(* CoDeSys 2.3.9.48 project: 20170405_WUR.pro *)
(* Version: 0.9 *)
(* Description: Project Distributie Automatisering *)
(* Libraries: Serial_Interface_01.lib 22.4.13 12:50:14, Util.lib 30.1.13 13:05:12, WagoLib787_01.lib 10.11.14 13:02:32, mod_com.lib 30.1.13 13:05:12, WagoConfigToolLIB.lib 30.1.13 13:05:12, C:\Program Files\WAGO Software\CODESYS V2.3\Targets\WAGO\Libraries\32_Bit\PowerMeasurement_495_02.lib*5.4.17 15:41:49, SysLibTime.lib 30.1.13 13:05:12, SerComm.lib 30.1.13 13:05:12, SysLibSockets.lib 22.5.14 16:16:32, SysLibFile.lib 30.1.13 13:05:12, C:\Program Files\WAGO Software\CODESYS V2.3\Targets\WAGO\Libraries\32_Bit\Ethernet.lib*5.4.17 15:41:49, SysLibMem.lib 30.1.13 13:05:12, SysLibSem.lib 30.1.13 13:05:12, SysLibRtc.lib 30.1.13 13:05:12, WagoLibEthernet_01.lib 1.4.15 14:24:28, WAGOLIBNTP.lib*19.8.11 14:53:14, Modb_l05.lib 13.5.15 10:30:08, SysLibDir.lib 30.1.13 13:05:12, C:\Program Files\WAGO Software\CODESYS V2.3\Targets\WAGO\Libraries\32_Bit\WAGO_Datalogger_02.lib*5.4.17 15:41:49, Wago_MBCFG_SERIAL_01.lib*1.4.15 14:24:28, Wago_MBCFG_COMMON_01.lib 1.4.15 14:24:28, Standard.lib 20.5.14 08:13:26, Iecsfc.lib 30.1.13 13:05:12, SYSLIBCALLBACK.LIB 30.1.13 13:05:12 *)

(* Task configuration *)
TASK WriteData (PRIORITY := 31); (* freewheeling *)
	WRITE_DATA();
END_TASK
TASK Measurements (PRIORITY := 1, INTERVAL := T#100ms);
	PQ_1();
END_TASK

(* Global variable list: Global_Variables *)
VAR_GLOBAL

	arMeasurementsGroup1					:	ARRAY[1.. iNumberMeasurementVar] OF REAL;
	arSystemState		AT %MW0			:	ARRAY[1.. iNumberSystemVar] OF REAL; 			(* Array containing all the system parameters. Values are accessable through modbus tcp starting from register 12288. REAL uses two registers per variable *)

END_VAR

VAR_GLOBAL CONSTANT

(* Read / write CSV-files *)
	iMaxParams			:	INT:=8;(* Number of Parameters per File *)
	gc_ParameterCount	:	INT:=1;(* Number of Values per Parameter *)
	gc_RawDataSize		:	UINT:=500; (* Raw data size for reading in file ASCII *)
	gcRowExcel			:	INT:=1;

	iNumberMeasurementVar	:	INT := 20;
	iNumberSystemVar			:	INT := 200;


END_VAR

VAR_GLOBAL PERSISTENT RETAIN

	CurrentRatioPQ1						:	WORD := 400;			(* Current transformer ratio, eg 5 A / 400 A *)
	CurrentRatioPQ2						:	WORD := 400;

END_VAR

(* Data type *)
TYPE typCSV :
STRUCT
	sDescription	:STRING;
	Parameter		:ARRAY[1..gc_ParameterCount] OF STRING;
END_STRUCT
END_TYPE

(* POU WRITE_CSV/WRITE_DATA, FBD *)
PROGRAM WRITE_DATA
VAR
	FB1				: FbDatalogger;
	xGo				: BOOL		:= TRUE;
	xTrigger			: BOOL;
	Channels			: ARRAY [1.. 80] OF typUserInput;
	Settings			: typConfigDatalogger;
	bDType			: BYTE := 1;
	xFirstCycle			: BOOL := TRUE;
	i: INT;

END_VAR
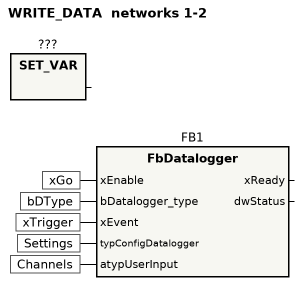
_FBD_ (* Function Block Diagram *)
NETWORK 1
	???:SET_VAR()
NETWORK 2
	FB1:FbDatalogger(xEnable: xGo, bDatalogger_type: bDType, xEvent: xTrigger, typConfigDatalogger: Settings, atypUserInput: Channels)
_END_FBD_
(* the same logic as Structured Text *)
(* Network 1: see the listing above *)
(* Network 2 *)
FB1(xEnable := xGo, bDatalogger_type := bDType, xEvent := xTrigger, typConfigDatalogger := Settings, atypUserInput := Channels);
END_PROGRAM
ACTION SET_VAR:
IF xFirstCycle THEN

	settings.bInterval					:= 3; 						(* 1 = hour, 2= minutes, 3 = seconds *)
	settings.iIntervalFactor			:= 5;						(* number of hours/minutes/seconds, depending on choice b.Interval *)
	settings.sFilename				:= 'Meetdata.csv';				(* Filename csv-file *)
	settings.sPath						:= '/media/sd/';				(* Path where the csv-file is stored *)
	settings.xAppendDate			:= TRUE;					(* When true, the date on the controller is added to the filename*)
	settings.xCyclicLogging			:= TRUE;					(* When true, information is stored cyclic on the controller/SD card *)

	Channels[1].xChannelExists		:= TRUE;
	Channels[1].sChannelName		:= 'PhaseCurrentl2';
	Channels[1].sUnit					:= 'A';
	Channels[1].rAlarmLowerLimit	:= -10000000;
	Channels[1].rAlarmUpperLimit	:= 10000000;

	Channels[2].xChannelExists		:= TRUE;
	Channels[2].sChannelName		:= 'VoltageV31';
	Channels[2].sUnit					:= 'V';
	Channels[2].rAlarmLowerLimit	:= -10000000;
	Channels[2].rAlarmUpperLimit	:= 10000000;

	Channels[3].xChannelExists		:= TRUE;
	Channels[3].sChannelName		:= 'Pactive';
	Channels[3].sUnit					:= 'W';
	Channels[3].rAlarmLowerLimit	:= -10000000;
	Channels[3].rAlarmUpperLimit	:= 10000000;

	Channels[4].xChannelExists		:= TRUE;
	Channels[4].sChannelName		:= 'Preactive';
	Channels[4].sUnit					:= 'VAr';;
	Channels[4].rAlarmLowerLimit	:= -10000000;
	Channels[4].rAlarmUpperLimit	:= 10000000;

	Channels[5].xChannelExists		:= TRUE;
	Channels[5].sChannelName		:= 'ShortCircuitDirectionA';
	Channels[5].sUnit					:= ' ';
	Channels[5].rAlarmLowerLimit	:= -10000000;
	Channels[5].rAlarmUpperLimit	:= 10000000;

	Channels[6].xChannelExists		:= TRUE;
	Channels[6].sChannelName		:= 'ShortCircuitDirectionB';
	Channels[6].sUnit					:= ' ';
	Channels[6].rAlarmLowerLimit	:= -10000000;
	Channels[6].rAlarmUpperLimit	:= 10000000;

	Channels[7].xChannelExists		:= TRUE;
	Channels[7].sChannelName		:= 'Phase1';
	Channels[7].sUnit					:= ' ';
	Channels[7].rAlarmLowerLimit	:= -10000000;
	Channels[7].rAlarmUpperLimit	:= 10000000;

	Channels[8].xChannelExists		:= TRUE;
	Channels[8].sChannelName		:= 'Phase2';
	Channels[8].sUnit					:=  ' ';
	Channels[8].rAlarmLowerLimit	:= -10000000;
	Channels[8].rAlarmUpperLimit	:= 10000000;

	Channels[9].xChannelExists		:= TRUE;
	Channels[9].sChannelName		:= 'Phase3';
	Channels[9].sUnit					:=  ' ';
	Channels[9].rAlarmLowerLimit	:= -10000000;
	Channels[9].rAlarmUpperLimit	:= 10000000;

	Channels[10].xChannelExists		:= TRUE;
	Channels[10].sChannelName		:= 'StatusRemoteSwitching';
	Channels[10].sUnit					:=  ' ';
	Channels[10].rAlarmLowerLimit	:= -10000000;
	Channels[10].rAlarmUpperLimit	:= 10000000;


	Channels[11].xChannelExists		:= TRUE;
	Channels[11].sChannelName		:= 'SwitchLoadBreaker';
	Channels[11].sUnit					:=  ' ';
	Channels[11].rAlarmLowerLimit	:= -10000000;
	Channels[11].rAlarmUpperLimit	:= 10000000;

	Channels[12].xChannelExists		:= TRUE;
	Channels[12].sChannelName		:= 'Bay3CurrentL1';
	Channels[12].sUnit					:=  'A ';
	Channels[12].rAlarmLowerLimit	:= -10000000;
	Channels[12].rAlarmUpperLimit	:= 10000000;

	Channels[13].xChannelExists		:= TRUE;
	Channels[13].sChannelName		:= 'Bay3CurrentL2';
	Channels[13].sUnit					:=  'A ';
	Channels[13].rAlarmLowerLimit	:= -10000000;
	Channels[13].rAlarmUpperLimit	:= 10000000;

	Channels[14].xChannelExists		:= TRUE;
	Channels[14].sChannelName		:= 'Bay3CurrentL3';
	Channels[14].sUnit					:=  'A ';
	Channels[14].rAlarmLowerLimit	:= -10000000;
	Channels[14].rAlarmUpperLimit	:= 10000000;

	Channels[15].xChannelExists		:= TRUE;
	Channels[15].sChannelName		:= 'Bay4CurrentL1';
	Channels[15].sUnit					:=  'A ';
	Channels[15].rAlarmLowerLimit	:= -10000000;
	Channels[15].rAlarmUpperLimit	:= 10000000;

	Channels[16].xChannelExists		:= TRUE;
	Channels[16].sChannelName		:= 'Bay4CurrentL2';
	Channels[16].sUnit					:=  'A ';
	Channels[16].rAlarmLowerLimit	:= -10000000;
	Channels[16].rAlarmUpperLimit	:= 10000000;

	Channels[17].xChannelExists		:= TRUE;
	Channels[17].sChannelName		:= 'Bay4CurrentL3';
	Channels[17].sUnit					:=  'A ';
	Channels[17].rAlarmLowerLimit	:= -10000000;
	Channels[17].rAlarmUpperLimit	:= 10000000;

	xFirstCycle := FALSE;

END_IF

	Channels[1].rValue			:= MBCFG_ModbusSlave.PhaseCurrenL2;
	Channels[2].rValue			:= MBCFG_ModbusSlave.VoltageV31;
	Channels[3].rValue			:= MBCFG_ModbusSlave.Pactive;
	Channels[4].rValue			:= MBCFG_ModbusSlave.Preactive;
	Channels[5].rValue			:= MBCFG_ModbusSlave.ShortCircuitA;
	Channels[6].rValue			:= MBCFG_ModbusSlave.ShortCircuitB;
	Channels[7].rValue			:= MBCFG_ModbusSlave.Phase1;
	Channels[8].rValue			:= MBCFG_ModbusSlave.Phase2;
	Channels[9].rValue			:= MBCFG_ModbusSlave.Phase3;
	Channels[10].rValue			:= MBCFG_ModbusSlave.StatusRemoteSwitching;
	Channels[11].rValue			:= MBCFG_ModbusSlave.SwitchLoadBreaker;
	Channels[12].rValue			:= PQ_1.arCurrent[1];
	Channels[13].rValue			:= PQ_1.arCurrent[2];
	Channels[14].rValue			:= PQ_1.arCurrent[3];
	Channels[15].rValue			:= PQ_2.arCurrent[1];
	Channels[16].rValue			:= PQ_2.arCurrent[2];
	Channels[17].rValue			:= PQ_2.arCurrent[3];





(* For-loop to set the channels to be written on the SD-card *)
END_ACTION

(* POU PQ/PQ_1, FBD *)
PROGRAM PQ_1
VAR
	abProcessImageInput	AT %IW48				: ARRAY[0..23] OF BYTE;
	abProcessImageOutput 	AT %QW48 			: ARRAY[0..23] OF BYTE;

	bToken										: BYTE;

	State_750_495 							: Fb_750_495_State;
		typ_750_495_State 						: typ_750_495_State;

	Configuration_750_495					: Fb_750_495_Configuration;
		typConfig_750_495						: typConfig_750_495;
		xReadyConfig								: BOOL;
		bFeedbackConfig							: BYTE;

	AC_Compact_01_750_495				: Fb_750_495_AC_Compact_01;
		rTotalActivePower							: REAL;
		rTotalReactivePower						: REAL;
		rTotalApparentPower						: REAL;
		rTotalPowerFactorPF						: REAL;
		rTotalActiveEnergy							: REAL;
		rTotalReactiveEnergy						: REAL;
		rTotalApparentEnergy						: REAL;
		rCurrentN									: REAL;
		xRotatingField								: BOOL;
		arCurrent									: ARRAY[1..3] OF REAL;
		axOvercurrent								: ARRAY[1..3] OF BOOL;
		arVoltage_L_N							: ARRAY[1..3] OF REAL;
		axUndervoltage							: ARRAY[1..3] OF BOOL;
		axOvervoltage								: ARRAY[1..3] OF BOOL;
		arActivePower								: ARRAY[1..3] OF REAL;
		arReactivePower							: ARRAY[1..3] OF REAL;
		arApparentPower							: ARRAY[1..3] OF REAL;
		arCosPhi									: ARRAY[1..3] OF REAL;
		arPowerFactorPF							: ARRAY[1..3] OF REAL;
		arFrequency								: ARRAY[1..3] OF REAL;
		axNoZero									: ARRAY[1..3] OF BOOL;
		axVoltSag									: ARRAY[1..3] OF BOOL;
		ai4Quadrant								: ARRAY[1..3] OF INT;

		xReadyCompact_01						: BOOL;
		abFeedbackCompact_01					: ARRAY[1..8] OF BYTE;


END_VAR
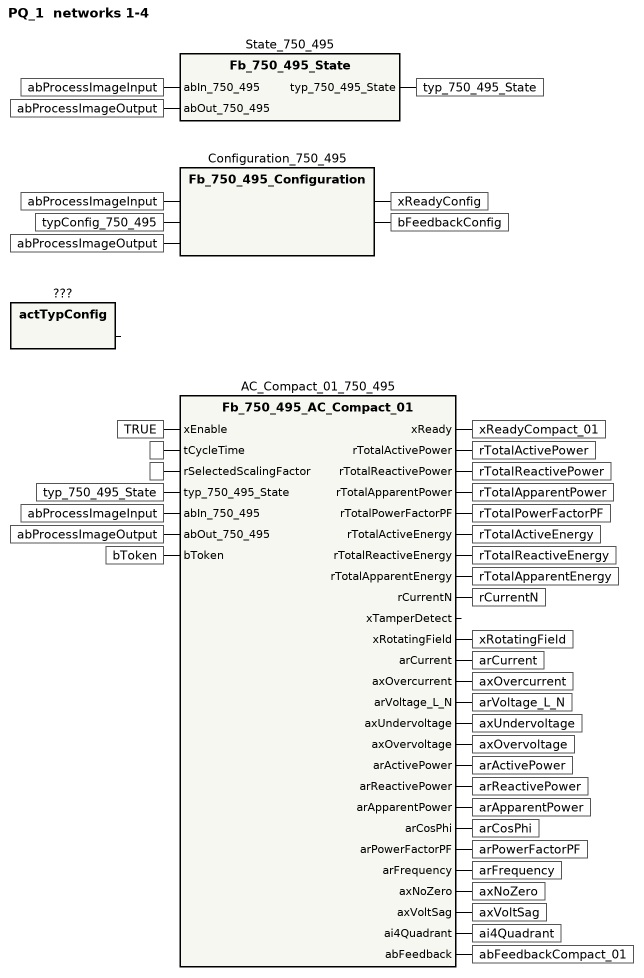
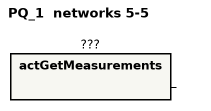
_FBD_ (* Function Block Diagram *)
NETWORK 1
	State_750_495:Fb_750_495_State(abIn_750_495: abProcessImageInput, abOut_750_495: abProcessImageOutput) => typ_750_495_State
NETWORK 2
	Configuration_750_495:Fb_750_495_Configuration(abProcessImageInput, typConfig_750_495, abProcessImageOutput, out 2 => bFeedbackConfig) => xReadyConfig
NETWORK 3
	???:actTypConfig()
NETWORK 4
	AC_Compact_01_750_495:Fb_750_495_AC_Compact_01(xEnable: TRUE, tCycleTime: , rSelectedScalingFactor: , typ_750_495_State: typ_750_495_State, abIn_750_495: abProcessImageInput, abOut_750_495: abProcessImageOutput, bToken: bToken, rTotalActivePower => rTotalActivePower, rTotalReactivePower => rTotalReactivePower, rTotalApparentPower => rTotalApparentPower, rTotalPowerFactorPF => rTotalPowerFactorPF, rTotalActiveEnergy => rTotalActiveEnergy, rTotalReactiveEnergy => rTotalReactiveEnergy, rTotalApparentEnergy => rTotalApparentEnergy, rCurrentN => rCurrentN, xRotatingField => xRotatingField, arCurrent => arCurrent, axOvercurrent => axOvercurrent, arVoltage_L_N => arVoltage_L_N, axUndervoltage => axUndervoltage, axOvervoltage => axOvervoltage, arActivePower => arActivePower, arReactivePower => arReactivePower, arApparentPower => arApparentPower, arCosPhi => arCosPhi, arPowerFactorPF => arPowerFactorPF, arFrequency => arFrequency, axNoZero => axNoZero, axVoltSag => axVoltSag, ai4Quadrant => ai4Quadrant, abFeedback => abFeedbackCompact_01) => xReadyCompact_01
NETWORK 5
	???:actGetMeasurements()
_END_FBD_
(* the same logic as Structured Text *)
(* Network 1 *)
State_750_495(abIn_750_495 := abProcessImageInput, abOut_750_495 := abProcessImageOutput);
typ_750_495_State := State_750_495.typ_750_495_State;
(* Network 2: see the listing above *)
(* Network 3: see the listing above *)
(* Network 4: see the listing above *)
(* Network 5: see the listing above *)
END_PROGRAM
ACTION actGetMeasurements:
arMeasurementsGroup1[1] := arVoltage_L_N[1];
arMeasurementsGroup1[2] := arVoltage_L_N[2];
arMeasurementsGroup1[3] := arVoltage_L_N[3];
arMeasurementsGroup1[4] := arCurrent[1];
arMeasurementsGroup1[5] := arCurrent[2];
arMeasurementsGroup1[6] := arCurrent[3];
END_ACTION
ACTION actTypConfig:
typConfig_750_495.typChannelConfig[1].xEnableUserScaling:= TRUE;
typConfig_750_495.typChannelConfig[1].wCurrentTransformerRatio :=CurrentRatioPQ1;

typConfig_750_495.typChannelConfig[2].xEnableUserScaling:= TRUE;
typConfig_750_495.typChannelConfig[2].wCurrentTransformerRatio :=CurrentRatioPQ1;

typConfig_750_495.typChannelConfig[3].xEnableUserScaling:= TRUE;
typConfig_750_495.typChannelConfig[3].wCurrentTransformerRatio :=CurrentRatioPQ1;

typConfig_750_495.xWriteConfig := TRUE;
END_ACTION

(* POU PLC_PRG, FBD *)
PROGRAM PLC_PRG
(*
  Function: 	Reading a CSV file
  Description: 	This project shows a functionblock which reads data from a CSV file into an array.
				Each line in the CSV contains a description and a real value.
				Each parameter  is terminated by CR LF.

---- Example CSV File -----

A_Value;245345
B_Value;0							
C_Value;8.3							
D_Value;-123439.3 						
E_Value;1						*)

VAR
	xLoad					: 	BOOL; (* Initiate load operation *)
	xSave					: 	BOOL; (* Initiate save operation *)
	sLoadStatus			: 	STRING; (* Feedback on load *)
	sSaveStatus			: 	STRING; (* Feedback on save *)
	ConfigData			: 	ARRAY [1..iMaxParams] OF  typCSV; (* Structure with the config data being loaded or saved *)
	sFileName			: 	STRING := 'config.csv'; (* Working Filename *)
	bSeperator 			: 	BYTE := 59; (* Semicolon (;) is the seperator between parameter and value. *)
	iError					: 	INT; (* Error Code for Save *)
	xWriteToSD			: 	BOOL := TRUE; (* User selectable location for file operation, on = 750-880 SD, off = internal flash *)
	sFilePath				: 	STRING; (* SD card is S:\, Internal Path is blank, but this points to the PLC folder *)
	sFilePath_Name		: 	STRING; (* Complete path + filename *)

	xReadFirstCycle		:	BOOL := TRUE;

	SetIPConfig				:	configToolFB;
	SetIP						:	configToolFB;
	SetSubnet					:	configToolFB;
	SetGateway				:	configToolFB;
	SetNTP					:	configToolFB;
	SetNTPEnable			:	configToolFB;
	SetSNMPName			:	configToolFB;
	SetSNMPDescription		:	configToolFB;
	SetSNMPLocation			:	configToolFB;
	SetSNMPContact			:	configToolFB;

	GetIPConfig				:	configToolFB;
	GetIP						:	configToolFB;
	GetSubnet					:	configToolFB;
	GetGateway				:	configToolFB;
	GetNTP					:	configToolFB;
	GetSNMPName			:	configToolFB;
	GetSNMPDescription		:	configToolFB;
	GetSNMPLocation		:	configToolFB;
	GetSNMPContact			:	configToolFB;
	GetFirmware				:	configToolFB;
	GetMACAddress			:	configToolFB;
	GetProjectDate			:	configToolFB;
	GetProjectDescription	:	configToolFB;
	GetProjectVersion			:	configToolFB;

	stSetIPConfigCallstring				:	STRING(80);
	stSetIPCallstring						:	STRING(80);
	stSetSubnetCallstring				:	STRING(80);
	stSetGatewayCallstring				:	STRING(80);
	stSetNTPCallstring					:	STRING(80);

	iSetIPConfigCallstringResult			:	INT;
	iSetIPCallstringResult				:	INT;
	iSetSubnetCallstringResult			:	INT;
	iSetGatewayCallstringResult			:	INT;
	iSetNTPCallstringResult				: 	INT;
	iSetNTPEnabledCallstringResult	:	INT;

	iGetIPConfigCallstringResult			:	INT;
	iGetIPCallstringResult				:	INT;
	iGetSubnetCallstringResult			:	INT;
	iGetGatewayCallstringResult			:	INT;
	iGetNTPCallstringResult				: 	INT;
	iGetNTPEnabledCallstringResult	:	INT;

	iGetFirmwareCallstringResult				:	INT;
	iGetMACAddressCallstringResult			:	INT;
	iGetProjectDateCallstringResult				:	INT;
	iGetProjectDescriptionCallstringResult		:	INT;
	iGetProjectVersionCallstringResult			:	INT;

	stGetIPConfigCallstring				:	STRING(80);
	stGetIPCallstring						:	STRING(80);
	stGetSubnetCallstring				:	STRING(80);
	stGetGatewayCallstring				:	STRING(80);
	stGetNTPCallstring					:	STRING(80);

	stSetIPConfigResult					:	STRING(80);
	stSetIPResult							:	STRING(80);
	stSetSubnetResult					:	STRING(80);
	stSetGatewayResult					:	STRING(80);
	stSetNTPResult						:	STRING(80);

	stGetIPConfigResult					:	STRING(80);
	stGetIPResult							:	STRING(80);
	stGetSubnetResult					:	STRING(80);
	stGetGatewayResult					:	STRING(80);
	stGetNTPResult						:	STRING(80);

	stSetSNMPNameDeviceCallstring					:	STRING(80);
	stSetSNMPDescriptionCallstring						:	STRING(80);
	stSetSNMPPhysicalLocationCallstring				:	STRING(80);
	stSetSNMPContactCallstring							:	STRING(80);

	stGetSNMPNameDeviceResult						:	STRING(80);
	stGetSNMPDescriptionResult						:	STRING(80);
	stGetSNMPPhysicalLocationResult					:	STRING(80);
	stGetSNMPContactResult							:	STRING(80);

	stGetFirmwareResult									:	STRING(80);
	stGetMACAddressResult								:	STRING(80);
	stGetProjectDateResult								:	STRING(80);
	stGetProjectDescriptionResult						:	STRING(80);
	stGetProjectVersionResult							:	STRING(80);

	iSetSNMPNameDeviceCallstringResult				:	INT;
	iSetSNMPDescriptionCallstringResult				:	INT;
	iSetSNMPPhysicalLocationCallstringResult			:	INT;
	iSetSNMPContactCallstringResult					:	INT;

	iGetSNMPNameDeviceCallstringResult				:	INT;
	iGetSNMPDescriptionCallstringResult				:	INT;
	iGetSNMPPhysicalLocationCallstringResult			:	INT;
	iGetSNMPContactCallstringResult					:	INT;

	CurrentTimeDate										:	STRING;

END_VAR
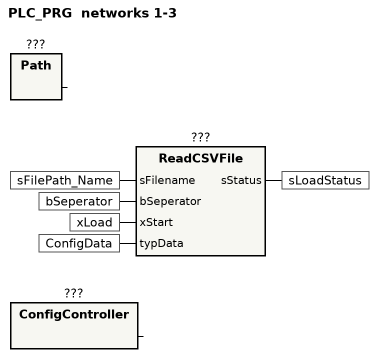
_FBD_ (* Function Block Diagram *)
NETWORK 1
	???:Path()
NETWORK 2
	???:ReadCSVFile(sFilename: sFilePath_Name, bSeperator: bSeperator, xStart: xLoad, typData: ConfigData) => sLoadStatus
NETWORK 3
	???:ConfigController()
_END_FBD_
END_PROGRAM
ACTION ConfigController:
IF xReadFirstCycle = TRUE THEN

	(*xLoad := TRUE;*)

	IF sLoadStatus = 'Data read OK' THEN
	
		(* Set Ethernet settings of controller *)
		
		(* Set static IP-Address*)
		
		
			SetIPConfig(
			bEnable:= TRUE,
			stCallString:= 'config_interfaces interface=X1 config-type=static state=enabled',
			stResultString=> stSetIPConfigResult,
			iFbResult=> iSetIPCallstringResult );
		
		(* Set IP-Address of controller *)
		
			stSetIPCallstring := CONCAT('config_interfaces interface X1 ip-address=',stIPAddressEthernet);
		
			SetIP(
			bEnable:= TRUE,
			stCallString:= stSetIPCallstring ,
			stResultString=> stSetIPResult,
			iFbResult=> iSetIPCallstringResult );
		
		(* Set Subnet-Address of controller *)
		
			stSetSubnetCallstring := CONCAT('config_interfaces interface X1 subnet-mask=',stIPAddressSubnet);
		
			SetSubnet(
			bEnable:= TRUE,
			stCallString:= stSetSubnetCallstring ,
			iFbResult=> iSetSubnetCallstringResult );
		
		(* Set Gateway-Address of controller *)
		
			stSetGatewayCallstring := CONCAT('config_default_gateway interface=X1 default-gateway-value=', stIPAddressGateway);
		
			SetGateway(
			bEnable:= TRUE,
			stCallString:= stSetGatewayCallstring ,
			iFbResult=> iSetGatewayCallstringResult );
		
		(* Set NTP-Address of controller *)
		
			SetNTPEnable(
			bEnable:= TRUE,
			stCallString:= 'config_sntp state=enabled' ,
			iFbResult=> iSetNTPEnabledCallstringResult );
		
			stSetNTPCallstring := CONCAT('config_sntp time-server=',stIPAddressNTP);
		
			SetNTP(
			bEnable:= TRUE,
			stCallString:= stSetNTPCallstring ,
			iFbResult=> iSetNTPCallstringResult );
		
		(* Set SNMP-configuration of the controller *)
		
		(* Set SNMP-description of the controller *)
		
			stSetSNMPDescriptionCallstring := CONCAT('config_snmp description=',stSNMPDescription);
		
			SetSNMPDescription(
			bEnable:= TRUE,
			stCallString:= stSetSNMPDescriptionCallstring,
			iFbResult=> iSetSNMPDescriptionCallstringResult );
		
		(* Set SNMP-name of the controller *)
		
			stSetSNMPNameDeviceCallstring := CONCAT('config_snmp device-name=',stSNMPNameDevice);
		
			SetSNMPName(
			bEnable:= TRUE,
			stCallString:= stSetSNMPNameDeviceCallstring,
			iFbResult=> iSetSNMPNameDeviceCallstringResult );
		
		(* Set SNMP-location of the controller *)

			stSetSNMPPhysicalLocationCallstring := CONCAT('config_snmp physical-location=',stSNMPPhysicalLocation);
		
			SetSNMPLocation(
			bEnable:= TRUE,
			stCallString:= stSetSNMPPhysicalLocationCallstring,
			iFbResult=> iSetSNMPPhysicalLocationCallstringResult);
		
		(* Set SNMP-contact information of the controller *)
		
			stSetSNMPContactCallstring := CONCAT('config_snmp contact=',stSNMPcontact);
		
			SetSNMPContact(
			bEnable:= TRUE,
			stCallString:= stSetSNMPContactCallstring,
			iFbResult=> iSetSNMPContactCallstringResult);
		
			xReadFirstCycle := FALSE;
			xLoad := FALSE;

	END_IF

END_IF

(* Get Ethernet settings of controller *)

(* Get IP-configuration of controller *)

	GetIPConfig(
	bEnable:= TRUE,
	stCallString:= 'get_eth_config X1 config-type' ,
	stResultString=> stGetIPConfigResult,
	iFbResult=> iGetIPConfigCallstringResult );

(* Get IP-Address of controller *)

	GetIP(
	bEnable:= TRUE,
	stCallString:= 'get_eth_config X1 ip-address' ,
	stResultString=> stGetIPResult,
	iFbResult=> iGetIPCallstringResult );

(* Get Subnet-Address of controller *)

	GetSubnet(
	bEnable:= TRUE,
	stCallString:= 'get_eth_config X1 subnet-mask' ,
	stResultString=> stGetSubnetResult,
	iFbResult=> iGetSubnetCallstringResult );

(* Get Gateway-Address of controller *)

	GetGateway(
	bEnable:= TRUE,
	stCallString:= 'get_eth_config X1 default-gateway' ,
	stResultString=> stGetGatewayResult,
	iFbResult=> iGetGatewayCallstringResult );

(* Get NTP-Address of controller *)

	GetNTP(
	bEnable:= TRUE,
	stCallString:= 'get_ntp_config time-server' ,
	stResultString=> stGetNTPResult,
	iFbResult=> iGetNTPCallstringResult );

(* Get SNMP-configuration of the controller *)

(* Get SNMP-description of the controller *)

	GetSNMPDescription(
	bEnable:= TRUE,
	stCallString:= 'get_snmp_data description',
	stResultString=> stGetSNMPDescriptionResult,
	iFbResult=> iGetSNMPDescriptionCallstringResult );

(* Get SNMP-description of the controller *)

	GetSNMPName(
	bEnable:= TRUE,
	stCallString:= 'get_snmp_data device-name',
	stResultString=> stGetSNMPNameDeviceResult,
	iFbResult=> iGetSNMPNameDeviceCallstringResult );

(* Get SNMP-location of the controller *)

	GetSNMPLocation(
	bEnable:= TRUE,
	stCallString:= 'get_snmp_data physical-location',
	stResultString=> stGetSNMPPhysicalLocationResult,
	iFbResult=> iGetSNMPPhysicalLocationCallstringResult);

(* Get SNMP-contact information of the controller *)

	GetSNMPContact(
	bEnable:= TRUE,
	stCallString:= 'get_snmp_data contact',
	stResultString=> stGetSNMPContactResult,
	iFbResult=> iGetSNMPContactCallstringResult);

(* Get Firmware information of the controller *)

	GetFirmware(
	bEnable:= TRUE,
	stCallString:= 'get_coupler_details firmware-revision',
	stResultString=> stGetFirmwareResult,
	iFbResult=> iGetFirmwareCallstringResult);

(* Get MAC-Address of the controller *)

	GetMACAddress(
	bEnable:= TRUE,
	stCallString:= 'get_actual_eth_config X1 mac-address',
	stResultString=> stGetMACAddressResult,
	iFbResult=> iGetMACAddressCallstringResult);

(* Get Project Date of the controller *)

	GetProjectDate(
	bEnable:= TRUE,
	stCallString:= 'get_rts_info project date',
	stResultString=> stGetProjectDateResult,
	iFbResult=> iGetProjectDateCallstringResult);

(* Get Project Description of the controller *)

	GetProjectDescription(
	bEnable:= TRUE,
	stCallString:= 'get_rts_info project description',
	stResultString=> stGetProjectDescriptionResult,
	iFbResult=> iGetProjectDescriptionCallstringResult);

(* Get Project version of the controller *)

	GetProjectVersion(
	bEnable:= TRUE,
	stCallString:= 'get_rts_info project version',
	stResultString=> stGetProjectVersionResult,
	iFbResult=> iGetProjectVersionCallstringResult);

	CurrentTimeDate := Date_Time();
END_ACTION
ACTION Path:
IF xWriteToSD THEN
	sFilePath := '/media/sd/';
ELSE
	sFilePath := '';
END_IF
sFilePath_Name := CONCAT(sFilePath, sFileName);
END_ACTION
ACTION SetParam:
	stIPAddressEthernet := ConfigData[1].Parameter[1];
	stIPAddressSubnet  := ConfigData[2].Parameter[1];
	stIPAddressGateway  := ConfigData[3].Parameter[1];
	stIPAddressNTP := ConfigData[4].Parameter[1];

	stSNMPNameDevice := ConfigData[5].Parameter[1];
	stSNMPDescription := ConfigData[6].Parameter[1];
	stSNMPPhysicalLocation := ConfigData[7].Parameter[1];
	stSNMPContact := ConfigData[8].Parameter[1];
END_ACTION

(* POU SD CARD/ReadCSVFile, ST *)
PROGRAM ReadCSVFile
VAR_INPUT
	sFilename		:STRING;
	bSeperator		:BYTE:=59;(*seperator semicolon:59=;*)
END_VAR
VAR_IN_OUT
	xStart			:BOOL;
	typData			:ARRAY [1..iMaxParams] OF  typCSV;
END_VAR
VAR_OUTPUT
	sStatus			:STRING;
END_VAR
VAR
	bEndOfFile		:BYTE:=13;
	FileIdent		:DWORD;
	rawdata			:ARRAY[0..gc_RawDataSize] OF BYTE;
	filesizev		:DINT;
	tempstring		:STRING;
	startposition	:INT;
	i				:INT;
	j				:INT;
	k				:INT;
END_VAR
IF xStart THEN
	FileIdent:=SysFileOpen(FileName:=sFilename, Mode:='r');
	IF fileident<>0 THEN
		SysFileRead(File:=Fileident, Buffer:=ADR(rawdata), Size:=SIZEOF(rawdata));
		filesizev:=SysFileGetSize(FileName:=sFilename);
		IF filesizev>gc_RawDataSize THEN
			filesizev:=gc_RawDataSize;
		END_IF
		SysFileClose(File:=fileident);(*this function is blocking*)
	ELSE
		sStatus:='File does not exist';
		xStart:=FALSE;
		RETURN;(*no such file available*)
	END_IF
(*copy data to typData array*)
	startposition:=0;
	i:=0;
	FOR j:=1 TO iMaxParams DO
		(*First value in dataset is of type DT. The following value is seperated by bSeperator*)
		WHILE rawdata[startposition+i]<>bSeperator DO
			i:=i+1;
		END_WHILE
		rawdata[startposition+i]:=0;
		MEMCPY(pSourceAddress:=ADR(rawdata[startposition]), pDestinationAddress:=ADR(tempstring), BytesToCopy:=i+1);
		typdata[j].sDescription:=tempstring;
		startposition:=startposition+i+1;
		i:=0;
		(*The parameter values are of type word. The following values are seperated by bSeperator*)
		FOR k:=1 TO gc_ParameterCount-1 DO
			WHILE rawdata[startposition+i]<>bSeperator DO
				i:=i+1;
			END_WHILE
			rawdata[startposition+i]:=0;
			MEMCPY(pSourceAddress:=ADR(rawdata[startposition]), pDestinationAddress:=ADR(tempstring), BytesToCopy:=i+1);
			typdata[j].Parameter[k]:=(tempstring);
			startposition:=startposition+i+1;
			i:=0;
		END_FOR
		(*Copying the last parameter from typ word. The data set is terminated by CR LF*)
		WHILE rawdata[startposition+i]<>bEndOfFile DO
			i:=i+1;
		END_WHILE
		rawdata[startposition+i]:=0;
		MEMCPY(pSourceAddress:=ADR(rawdata[startposition]), pDestinationAddress:=ADR(tempstring), BytesToCopy:=i+1);
		typdata[j].Parameter[k]:=(tempstring);
		startposition:=startposition+i+2;(*The data set is terminated by CR LF(13,10)*)
		i:=0;
	END_FOR
(*copy data to typData array finished*)
	sStatus:='Data read OK';
	xStart:=FALSE;
END_IF
END_PROGRAM

(* POU MAIN, ST *)
PROGRAM MAIN
VAR
	i: INT;
END_VAR
FOR i := 1 TO iNumberSystemVar DO

	IF i <= iNumberMeasurementVar THEN

		arSystemState[i] := arMeasurementsGroup1[i];

	END_IF

	IF i > iNumberMeasurementVar AND  i <= 2*iNumberMeasurementVar THEN

		arSystemState[i] := arMeasurementsGroup1[i];

	END_IF

END_FOR
END_PROGRAM

(* POU Configuration/MODBUS_CONFIGURATION, ST *)
PROGRAM MODBUS_CONFIGURATION        
VAR                                
END_VAR                            
(*                                 
   <?xml version="1.0" encoding="UTF-16" standalone="yes"?>
<network xml_structure_version="1" xml_feature_version="1">
	<generator_settings minRTUTaskCycleTimeMs="100" minEthaskCycleTimeMs="5" ethSlaveMultiplier="0.1" rtuInterfaceMultiplier="0.1" taskGeneration="true"/>
	<master_interface type="serial" name="Configuration Root Node" com_port="2" baudrate="9600" databits="8" stopbits="1" parity="even" hwtype="RS485" flow_control="Xon/Xoff" asciimode="false" expanded="true">
		<mb_slave comment="" name="ModbusSlave" expanded="true" type="generic">
			<mb_connection type="serial" unitid="1" request_delay_ms="0" response_timeout_ms="1000"/>
			<generic_vars comment="" expanded="true">
				<generic_var data_type="REAL">
					<generic_params name="PhaseCurrenL2" comment="" expanded="false" mb_iotype="unused" mb_access="ro" var_byteorder="B3B4B1B2"/>
					<mb_address explicitAccess="false" FCRead="3" FCWrite="0" ReadMBAddress="20002" WriteMBAddress="0" ReadBitOffset="0" WriteBitOffset="0"/>
				</generic_var>
				<generic_var data_type="REAL">
					<generic_params name="VoltageV31" comment="" expanded="true" mb_iotype="unused" mb_access="ro" var_byteorder="B3B4B1B2"/>
					<mb_address explicitAccess="false" FCRead="3" FCWrite="0" ReadMBAddress="20012" WriteMBAddress="0" ReadBitOffset="0" WriteBitOffset="0"/>
				</generic_var>
				<generic_var data_type="REAL">
					<generic_params name="Pactive" comment="" expanded="true" mb_iotype="unused" mb_access="ro" var_byteorder="B3B4B1B2"/>
					<mb_address explicitAccess="false" FCRead="3" FCWrite="0" ReadMBAddress="20048" WriteMBAddress="0" ReadBitOffset="0" WriteBitOffset="0"/>
				</generic_var>
				<generic_var data_type="UINT">
					<generic_params name="ShortCircuitA" comment="" expanded="false" mb_iotype="unused" mb_access="ro" var_byteorder="B1B2B3B4"/>
					<mb_address explicitAccess="false" FCRead="3" FCWrite="0" ReadMBAddress="21002" WriteMBAddress="0" ReadBitOffset="0" WriteBitOffset="0"/>
				</generic_var>
				<generic_var data_type="UINT">
					<generic_params name="ShortCircuitB" comment="" expanded="true" mb_iotype="unused" mb_access="ro" var_byteorder="B1B2B3B4"/>
					<mb_address explicitAccess="false" FCRead="3" FCWrite="0" ReadMBAddress="21003" WriteMBAddress="0" ReadBitOffset="0" WriteBitOffset="0"/>
				</generic_var>
				<generic_var data_type="REAL">
					<generic_params name="Preactive" comment="" expanded="true" mb_iotype="unused" mb_access="ro" var_byteorder="B3B4B1B2"/>
					<mb_address explicitAccess="false" FCRead="3" FCWrite="0" ReadMBAddress="20050" WriteMBAddress="0" ReadBitOffset="0" WriteBitOffset="0"/>
				</generic_var>
				<generic_var data_type="UINT">
					<generic_params name="Phase1" comment="" expanded="false" mb_iotype="unused" mb_access="ro" var_byteorder="B1B2B3B4"/>
					<mb_address explicitAccess="false" FCRead="3" FCWrite="0" ReadMBAddress="21036" WriteMBAddress="0" ReadBitOffset="0" WriteBitOffset="0"/>
				</generic_var>
				<generic_var data_type="UINT">
					<generic_params name="Phase2" comment="" expanded="false" mb_iotype="unused" mb_access="ro" var_byteorder="B1B2B3B4"/>
					<mb_address explicitAccess="false" FCRead="3" FCWrite="0" ReadMBAddress="21037" WriteMBAddress="0" ReadBitOffset="0" WriteBitOffset="0"/>
				</generic_var>
				<generic_var data_type="UINT">
					<generic_params name="Phase3" comment="" expanded="false" mb_iotype="unused" mb_access="ro" var_byteorder="B1B2B3B4"/>
					<mb_address explicitAccess="false" FCRead="3" FCWrite="0" ReadMBAddress="21038" WriteMBAddress="0" ReadBitOffset="0" WriteBitOffset="0"/>
				</generic_var>
				<generic_var data_type="UINT">
					<generic_params name="StatusRemoteSwitching" comment="" expanded="false" mb_iotype="unused" mb_access="ro" var_byteorder="B1B2B3B4"/>
					<mb_address explicitAccess="false" FCRead="3" FCWrite="0" ReadMBAddress="23000" WriteMBAddress="0" ReadBitOffset="0" WriteBitOffset="0"/>
				</generic_var>
				<generic_var data_type="UINT">
					<generic_params name="SwitchLoadBreaker" comment="" expanded="true" mb_iotype="unused" mb_access="wo" var_byteorder="B1B2B3B4"/>
					<mb_address explicitAccess="false" FCRead="0" FCWrite="6" ReadMBAddress="0" WriteMBAddress="23100" ReadBitOffset="0" WriteBitOffset="0"/>
				</generic_var>
			</generic_vars>
		</mb_slave>
	</master_interface>
</network>
                              
*)                                 
;                                  
END_PROGRAM

(* POU SD CARD/WriteCSVFile, ST *)
PROGRAM WriteCSVFile
(* 	This function block Writes the contents of the data structure to a CSV File

	Required Libraries:
		Standard.lib
		SysLibFile.lib
*)
VAR_INPUT
	sFILENAME 		:STRING(80); (* Filename to store data to (e.g. 'config.csv' 		*)
	typData			:ARRAY [1..iMaxParams] OF typCSV;
	bSeperator		:BYTE :=59;	(* Seperator semicolon:59=;*)
END_VAR
VAR_IN_OUT
	xStart 			:BOOL;	(* Set TRUE to write data, set False to stop.		 *)
END_VAR
VAR_OUTPUT
	sStatus			:STRING;
	iError 			:INT;	(* 00 : Normal Operation	*)
							(* 90 : Can't Open File 	*)
							(* 91 : Can't Close File 	*)
							(* 92 : Can't Write to File 	*)
END_VAR
VAR
	FileOpen		:BOOL := FALSE;
	handle			:DWORD;
	Mode			:STRING[20] := 'rw'; (* read/write *)
	DataString 		:STRING(80);
	i				:INT;
END_VAR
IF xStart THEN
	sStatus := 'Try to open file';
	IF NOT FileOpen THEN
		(* Open File *)
		handle := SysFileOpen(sFileName, Mode);
		IF handle > 0 THEN
			FileOpen := TRUE;
			sStatus := 'File Open OK.';
		ELSE
			iERROR := 90; (* Could not open file. *)
			sStatus := 'Could not open file.';
		END_IF
	END_IF
	
	IF FileOpen THEN
		FOR i := 1 TO iMaxParams DO
				DataString := TypData[i].sDescription;
				DataString := CONCAT(DataString,ASCIIBYTE_TO_STRING(bSeperator));
				DataString := CONCAT(DataString,(TypData[i].Parameter[1]));
	
				DataString := CONCAT(DataString,ASCIIBYTE_TO_STRING(13)); (* CR *)
				DataString := CONCAT(DataString,ASCIIBYTE_TO_STRING(10)); (* LF *)
				(* Write string to file *)
				IF SysFileWrite(handle, ADR(DataString), LEN(DataString)) = 0 THEN
					iERROR := 92; (* Could not write to file *)
					sStatus := 'Could not write file.';
				END_IF
		END_FOR
	END_IF
	
	IF FileOpen THEN
		(* Close file *)
		IF SysFileClose(handle) THEN
			FileOpen := FALSE;
			sStatus := 'File Saved.';
		ELSE
			iERROR := 91; (* Could not close file *)
			sStatus := 'Could not close file.';
		END_IF
		xStart := FALSE;
	END_IF
END_IF
END_PROGRAM
